PROGRAM prgComEffIO
VAR
	fbCom		: FB_MqttCommunicator_V3;
END_VAR

fbCom(
	bConnect:= TRUE, 
	strAuthKey:=  'BMS99299754422' , 
	sUserName:= '673dfecd-87ae-41b4-adc6-bf4a9ec1d31b', 
	sUserPassword:= '6bd7bf44-8c7f-4537-ab63-8e71aabc2a94', 
	eSavePositionCertificate:= eSavePositionOnPLC.ePostionHardDisk, 
	time_HeartBeat_sec := T#15S,
	bConnected=> , 
	bError=> , 
	hrErrorCode=> , 
	eConnectionState=> , 
	eErrorMessage_Out=> );
	
(*old 
	sUserName:= '21f91cb5-8a07-4d3e-84c2-8bec390be0dd', 
	sUserPassword:= '26145dc9-e42c-4011-8f9c-6df6dcfb29f6', 
*)

END_PROGRAM

(* stored: Version 1.1.0.1, ProductVersion 3.1.4024.12
   POU prgComEffIO: Id {cbcd318b-bf51-484c-bcaa-d6efcdf43fe3}, SpecialFunc None *)
